{attribute 'qualified_only'}
VAR_GLOBAL
	AxisX_Feedback		: AxisFeedback;
	AxisY_Feedback		: AxisFeedback;
	AxisZ_Feedback		: AxisFeedback;
END_VAR

(* stored: Version 1.1.0.1, ProductVersion 3.1.4024.10
   GVL Feedback: Id {0fea718b-4e5e-4198-8b41-16d0c7c7591b} *)
